TYPE ST_Euchner_MSM_IN :
STRUCT
	///SM_I_S1 | Nothalt
	bSM_I_S1: BOOL;
	///SM_I_S2 | Taster beleuchtet
	bSM_I_S2: BOOL;
	///SM_I_S3 | Taster beleuchtet
	bSM_I_S3: BOOL;
	///SM_E_S1 | Fehler Sx
	bSM_E_S1: BOOL;
END_STRUCT
END_TYPE

(* stored: Version 1.1.0.1, ProductVersion 3.1.4024.12
   DUT ST_Euchner_MSM_IN: Id {2a0618c7-3735-4579-94b5-93ec12e3c710} *)
